Universal Robots URScript: KZXD.script

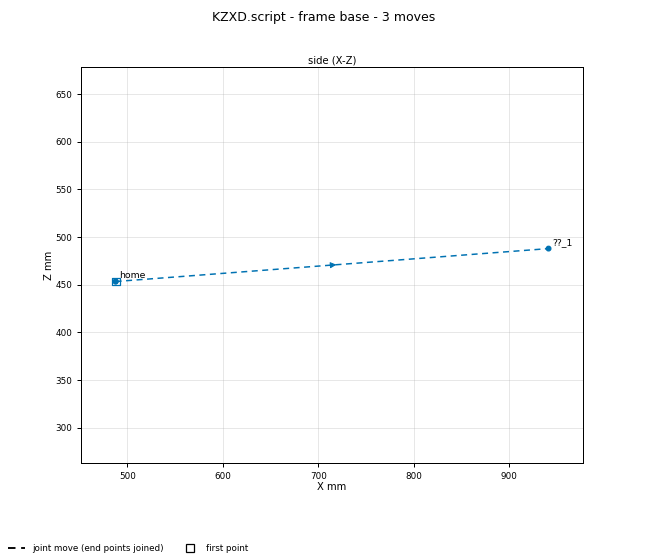
[picture p0: tool path of KZXD.script in frame base, 3 of 6 moves have a stored position in this frame; points joined in program order, loops and branches not executed]
def KZXD():
  set_tcp(p[0.0,0.0,0.0,0.0,0.0,0.0])
  set_payload(3.5)
  set_safety_mode_transition_hardness(1)
  set_standard_analog_input_domain(0, 1)
  set_standard_analog_input_domain(1, 1)
  set_tool_analog_input_domain(0, 1)
  set_tool_analog_input_domain(1, 1)
  set_analog_outputdomain(0, 0)
  set_analog_outputdomain(1, 0)
  set_input_actions_to_default()
  set_gravity([0.0, 0.0, 9.82])
  set_tool_voltage(0)
  global cnt_1=0
  $ 1 "机器人程序"
  $ 2 "设置 DO[1]=关"
  set_standard_digital_out(1, False)
  $ 3 "MoveJ"
  $ 4 "home"
  movej(get_inverse_kin(p[.487593461935, .103241290240, .453443983193, -1.735600206815, .715822306184, -1.707857722324], qnear=[-3.3179641405688685, -1.6227229277240198, 2.403541326522827, -3.927544895802633, -1.360473934804098, -0.7436946074115198]), a=1.3962634015954636, v=1.0471975511965976)
  $ 5 "路点_1"
  movej(get_inverse_kin(p[.941573521855, .103268444059, .487983012623, -2.846964411227, 1.245649618149, .043906619583], qnear=[-3.2174609343158167, -1.1385186354266565, 1.320655345916748, -1.740119759236471, -1.5344646612750452, -0.8131955305682581]), a=1.3962634015954636, v=1.0471975511965976)
  $ 6 "等待: 20.0"
  sleep(20.0)
  $ 7 "循环 3 次数"
  u24490u29615_1 = 0
  while (u24490u29615_1 < 3):
    $ 8 "设置 DO[0]=开"
    set_standard_digital_out(0, True)
    $ 9 "托盘"
    u20301u23039_1 = interpolate_pose(p[1.060103528391, .475452561391, .177812637361, -2.887209323466, 1.233162646416, .045049015855],p[1.060076988130, -.612279209413, .166250523809, -2.887264695428, 1.233098884872, .045019165403], cnt_1/2.0)
    if (cnt_1 >= 2):
      cnt_1 = 0
    else:
      cnt_1 = cnt_1 + 1
    end
    $ 14 "方式"
    movel(pose_trans(u20301u23039_1, pose_trans(pose_inv(p[1.060105201597, .475439993612, .177830662408, -2.887194699037, 1.233095164503, .045000736205]),p[1.060150374785, .475394959392, .237069360704, -2.887040274070, 1.233198936195, .044702528655])), a=1.2, v=0.25)
    $ 15 "模式点_1"
    movel(u20301u23039_1, a=1.2, v=0.25)
    $ 16 "设置"
    $ 18 "退出"
    movel(pose_trans(u20301u23039_1, pose_trans(pose_inv(p[1.060105201597, .475439993612, .177830662408, -2.887194699037, 1.233095164503, .045000736205]),p[1.060139884516, .475412014234, .237065340310, -2.887053064589, 1.233103529562, .044805787690])), a=1.2, v=0.25)
    u24490u29615_1 = u24490u29615_1 + 1
  end
  $ 19 "设置 DO[0]=关"
  set_standard_digital_out(0, False)
  $ 21 "MoveJ"
  $ 22 "路点_2"
  movej(get_inverse_kin(p[.487599235313, .103199775775, .453463312105, -1.735594233069, .715853107176, -1.707908120260], qnear=[-3.3180599848376673, -1.622758690510885, 2.403529167175293, -3.927509133015768, -1.3604257742511194, -0.7437065283404749]), a=1.3962634015954636, v=1.0471975511965976)
  $ 23 "设置 DO[1]=开"
  set_standard_digital_out(1, True)
end
